{attribute addProperty BoxType "EL2521-1001-0000"}
{attribute addProperty Id "InputsAT %I*Inputs_44EC503A2430OutputsAT %Q*Outputs_C13D2F242430WcStateAT %I*WcState_98A4DF7520.250InfoDataAT %I*InfoData_BC63D37F80100"}
{attribute addProperty CRC "875563102"}
{attribute addProperty SizeInBites "130"}
{attribute addProperty SizeInBytes "16.25"}
TYPE EL2521_30466534 :
STRUCT
	{attribute addProperty Name "Inputs"}
	Inputs : Inputs_44EC503A;
	{attribute addProperty Name "Outputs"}
	Outputs : Outputs_C13D2F24;
	{attribute addProperty Name "WcState"}
	WcState : WcState_98A4DF75;
	{attribute addProperty Name "InfoData"}
	InfoData : InfoData_BC63D37F;
END_STRUCT
END_TYPE

(* stored: Version 1.2.0.0, ProductVersion 3.1.4024.9
   DUT EL2521_30466534: Id {30b4d8df-1cc1-41de-aab9-c5d01a6eb715} *)
